Fanuc TP program (LS listing): JOB_VAR_SETUP.LS

/PROG  JOB_VAR_SETUP
/ATTR
OWNER		= MNEDITOR;
COMMENT		= "";
PROG_SIZE	= 12065;
CREATE		= DATE 19-06-21  TIME 11:36:36;
MODIFIED	= DATE 25-04-24  TIME 17:11:18;
FILE_NAME	= JOB_VAR_;
VERSION		= 0;
LINE_COUNT	= 453;
MEMORY_SIZE	= 12577;
PROTECT		= READ_WRITE;
TCD:  STACK_SIZE	= 0,
      TASK_PRIORITY	= 50,
      TIME_SLICE	= 0,
      BUSY_LAMP_OFF	= 0,
      ABORT_REQUEST	= 0,
      PAUSE_REQUEST	= 0;
DEFAULT_GROUP	= 1,*,*,*,*;
CONTROL_CODE	= 00000000 00000000;
/APPL

AUTO_SINGULARITY_HEADER;
  ENABLE_SINGULARITY_AVOIDANCE   : TRUE;
/MN
   1:  !--------------------------- ;
   2:  !Define the following run-time ;
   3:  !System variables, based on specs ;
   4:  !R[105]=AR[1]=100, 2By3 Sheet ;
   5:  !R[105]=AR[1]=200, 3By4 Sheet ;
   6:  !R[105]=AR[1]=300, 5By7 Sheet ;
   7:  !R[105]=AR[1]=400, 4By6 Sheet ;
   8:  !--------------------------- ;
   9:  !Input AR[1] Determines Setup ;
  10:  R[105]=AR[1]    ;
  11:  SELECT R[105]=100,JMP LBL[100] ;
  12:  !--------------------------- ;
  13:  !3By4 Sheet, 36 piece per Infeed ;
  14:  !Table Point, 36 Per level ;
  15:  !--------------------------- ;
  16:         =200,JMP LBL[200] ;
  17:  !--------------------------- ;
  18:  !3By4 Sheet Mandrel, 36 piece per ;
  19:  !Table Point, 36 Per level ;
  20:  !--------------------------- ;
  21:         =210,JMP LBL[210] ;
  22:  !--------------------------- ;
  23:  !3By4 , 36 piece per ;
  24:  !BOX, 36 Per level ;
  25:  !--------------------------- ;
  26:         =220,JMP LBL[220] ;
  27:  !--------------------------- ;
  28:  !5By7 Sheet, 35 piece per tray ;
  29:  !Table Point, 35 Per tray ;
  30:  !--------------------------- ;
  31:         =300,JMP LBL[300] ;
  32:  !--------------------------- ;
  33:  !4By6 INF, 144 piece per table ;
  34:  !4By9 OTF, 144 piece per table ;
  35:  !--------------------------- ;
  36:         =400,JMP LBL[400] ;
  37:  !--------------------------- ;
  38:  !Bar Feed, Outfeed Only ;
  39:  !4By9 OTF, 144 piece per table ;
  40:  !--------------------------- ;
  41:         =410,JMP LBL[410] ;
  42:  !--------------------------- ;
  43:  !4By6 INF, 144 piece per table ;
  44:  !6By8 OTF, 144 piece per table ;
  45:  !--------------------------- ;
  46:         =450,JMP LBL[450] ;
  47:  !--------------------------- ;
  48:  !6By8 OTF, 144 piece per table ;
  49:  !--------------------------- ;
  50:         =470,JMP LBL[470] ;
  51:  !--------------------------- ;
  52:  !3By4 Sheet, metal plate 12 piece ;
  53:  !Table Point, 36 Per tray ;
  54:  !--------------------------- ;
  55:         =500,JMP LBL[500] ;
  56:  !--------------------------- ;
  57:  !3By4 Sheet, 12 piece per tray ;
  58:  !Table Point, 72 Per level ;
  59:  !--------------------------- ;
  60:         =600,JMP LBL[600] ;
  61:  !--------------------------- ;
  62:  !Pallet data from Karel program ;
  63:  !--------------------------- ;
  64:         =900,JMP LBL[900] ;
  65:  !--------------------------- ;
  66:  !Beginning of Logic Program ;
  67:  !--------------------------- ;
  68:  LBL[100] ;
  69:  !--------------------------- ;
  70:  !2By3 Sheet, 6 piece per Infeed ;
  71:  !Table Point, 18 Per level ;
  72:  !--------------------------- ;
  73:  !1st: Infeed Row Offset ;
  74:  R[80]=191    ;
  75:  !2nd: Infeed Column Offset ;
  76:  R[81]=191    ;
  77:  !3rd: Infeed Division Offset ;
  78:  R[82]=2    ;
  79:  !4th: Infeed Modulus Offset ;
  80:  R[83]=2    ;
  81:  !5th: Infeed # of Pieces Per ;
  82:  !P[1], ie. One Level 3*(#) ;
  83:  !P[1] segnment of table, R[84] ;
  84:  R[84]=18    ;
  85:  !6th: Outfeed Row Offset ;
  86:  R[90]=191    ;
  87:  !7th: Outfeed Column Offset ;
  88:  R[91]=191    ;
  89:  !8th: Outfeed Division Offset ;
  90:  R[92]=2    ;
  91:  !9th: Outfeed Modulus Offset ;
  92:  R[93]=2    ;
  93:  !10th: Outfeed # of Pieces Per ;
  94:  !P[1], ie. One Level 3*(#) ;
  95:  !P[1] segnment of table, R[94] ;
  96:  R[94]=18    ;
  97:  JMP LBL[5000] ;
  98:   ;
  99:  LBL[200] ;
 100:  !--------------------------- ;
 101:  !3By4 Sheet, 12 piece per Infeed ;
 102:  !Table Point, 36 Per level ;
 103:  !--------------------------- ;
 104:  !1st: Infeed Row Offset ;
 105:  R[80]=140    ;
 106:  !2nd: Infeed Column Offset ;
 107:  R[81]=140    ;
 108:  !3rd: Infeed Division Offset ;
 109:  R[82]=3    ;
 110:  !4th: Infeed Modulus Offset ;
 111:  R[83]=3    ;
 112:  !5th: Infeed # of Pieces Per ;
 113:  !P[1], ie. One Level 3*(#) ;
 114:  !P[1] segnment of table, R[84] ;
 115:  R[84]=36    ;
 116:  !6th: Outfeed Row Offset ;
 117:  R[90]=130    ;
 118:  !7th: Outfeed Column Offset ;
 119:  R[91]=130    ;
 120:  !8th: Outfeed Division Offset ;
 121:  R[92]=3    ;
 122:  !9th: Outfeed Modulus Offset ;
 123:  R[93]=3    ;
 124:  !10th: Outfeed # of Pieces Per ;
 125:  !P[1], ie. One Level 3*(#) ;
 126:  !P[1] segnment of table, R[94] ;
 127:  R[94]=36    ;
 128:  JMP LBL[5000] ;
 129:   ;
 130:  LBL[210] ;
 131:  !--------------------------- ;
 132:  !3By4 Sheet, 12 piece per Infeed ;
 133:  !Table Point, 36 Per level ;
 134:  !metal plate, for mandrel ;
 135:  !--------------------------- ;
 136:  !1st: Infeed Row Offset ;
 137:  R[80]=126.9    ;
 138:  !2nd: Infeed Column Offset ;
 139:  R[81]=126.8    ;
 140:  !3rd: Infeed Division Offset ;
 141:  R[82]=3    ;
 142:  !4th: Infeed Modulus Offset ;
 143:  R[83]=3    ;
 144:  !5th: Infeed # of Pieces Per ;
 145:  !P[1], ie. One Level 3*(#) ;
 146:  !P[1] segnment of table, R[84] ;
 147:  R[84]=36    ;
 148:  !6th: Outfeed Row Offset ;
 149:  R[90]=130    ;
 150:  !7th: Outfeed Column Offset ;
 151:  R[91]=131    ;
 152:  !8th: Outfeed Division Offset ;
 153:  R[92]=3    ;
 154:  !9th: Outfeed Modulus Offset ;
 155:  R[93]=3    ;
 156:  !10th: Outfeed # of Pieces Per ;
 157:  !P[1], ie. One Level 3*(#) ;
 158:  !P[1] segnment of table, R[94] ;
 159:  R[94]=36    ;
 160:  JMP LBL[5000] ;
 161:  !--------------------------- ;
 162:  LBL[220] ;
 163:  !--------------------------- ;
 164:  !3By4 BOX, 12 piece per Infeed ;
 165:  !Table Point, 36 Per level ;
 166:  !--------------------------- ;
 167:  !1st: Infeed Row Offset ;
 168:  R[80]=127.2    ;
 169:  !2nd: Infeed Column Offset ;
 170:  R[81]=128.1    ;
 171:  !3rd: Infeed Division Offset ;
 172:  R[82]=3    ;
 173:  !4th: Infeed Modulus Offset ;
 174:  R[83]=3    ;
 175:  !5th: Infeed # of Pieces Per ;
 176:  !P[1], ie. One Level 3*(#) ;
 177:  !P[1] segnment of table, R[84] ;
 178:  R[84]=36    ;
 179:  !6th: Outfeed Row Offset ;
 180:  R[90]=127    ;
 181:  !7th: Outfeed Column Offset ;
 182:  R[91]=127    ;
 183:  !8th: Outfeed Division Offset ;
 184:  R[92]=3    ;
 185:  !9th: Outfeed Modulus Offset ;
 186:  R[93]=3    ;
 187:  !10th: Outfeed # of Pieces Per ;
 188:  !P[1], ie. One Level 3*(#) ;
 189:  !P[1] segnment of table, R[94] ;
 190:  R[94]=36    ;
 191:  JMP LBL[5000] ;
 192:   ;
 193:  LBL[300] ;
 194:  !--------------------------- ;
 195:  !5By7 Sheet, 35 piece per Infeed ;
 196:  !Table Point, 105 Per level ;
 197:  !--------------------------- ;
 198:  !1st: Infeed Row Offset ;
 199:  R[80]=76.2    ;
 200:  !2nd: Infeed Column Offset ;
 201:  R[81]=76.2    ;
 202:  !3rd: Infeed Division Offset ;
 203:  R[82]=5    ;
 204:  !4th: Infeed Modulus Offset ;
 205:  R[83]=5    ;
 206:  !5th: Infeed # of Pieces Per ;
 207:  !P[1], ie. One Level 3*(#) ;
 208:  !P[1] segnment of table, R[84] ;
 209:  R[84]=105    ;
 210:  !6th: Outfeed Row Offset ;
 211:  R[90]=130    ;
 212:  !7th: Outfeed Column Offset ;
 213:  R[91]=130    ;
 214:  !8th: Outfeed Division Offset ;
 215:  R[92]=3    ;
 216:  !9th: Outfeed Modulus Offset ;
 217:  R[93]=3    ;
 218:  !10th: Outfeed # of Pieces Per ;
 219:  !P[1], ie. One Level 3*(#) ;
 220:  !P[1] segnment of table, R[94] ;
 221:  R[94]=36    ;
 222:  JMP LBL[5000] ;
 223:   ;
 224:  LBL[400] ;
 225:  !--------------------------- ;
 226:  !4By6 INF, 24 piece per tray, 144 ;
 227:  !4By9 OTF, 36 piece per tray, 144 ;
 228:  !--------------------------- ;
 229:  !1st: Infeed Row Offset ;
 230:  R[80]=101.6    ;
 231:  !2nd: Infeed Column Offset ;
 232:  R[81]=101.8    ;
 233:  !3rd: Infeed Division Offset ;
 234:  R[82]=4    ;
 235:  !4th: Infeed Modulus Offset ;
 236:  R[83]=4    ;
 237:  !5th: Infeed # of Pieces Per ;
 238:  !P[1], ie. One Level 3*(#) ;
 239:  !P[1] segnment of table, R[84] ;
 240:  R[84]=144    ;
 241:  !6th: Outfeed Row Offset ;
 242:  R[90]=63.5    ;
 243:  !7th: Outfeed Column Offset ;
 244:  R[91]=63    ;
 245:  !8th: Outfeed Division Offset ;
 246:  R[92]=4    ;
 247:  !9th: Outfeed Modulus Offset ;
 248:  R[93]=4    ;
 249:  !10th: Outfeed # of Pieces Per ;
 250:  !P[1], ie. One Level 3*(#) ;
 251:  !P[1] segnment of table, R[94] ;
 252:  R[94]=144    ;
 253:  JMP LBL[5000] ;
 254:   ;
 255:  LBL[410] ;
 256:  !--------------------------- ;
 257:  !4By9 OTF, 36 piece per tray, 144 ;
 258:  !--------------------------- ;
 259:  !1st: Infeed Row Offset ;
 260:  R[80]=101.6    ;
 261:  !2nd: Infeed Column Offset ;
 262:  R[81]=101.8    ;
 263:  !3rd: Infeed Division Offset ;
 264:  R[82]=4    ;
 265:  !4th: Infeed Modulus Offset ;
 266:  R[83]=4    ;
 267:  !5th: Infeed # of Pieces Per ;
 268:  !P[1], ie. One Level 3*(#) ;
 269:  !P[1] segnment of table, R[84] ;
 270:  R[84]=144    ;
 271:  !6th: Outfeed Row Offset ;
 272:  R[90]=63.5    ;
 273:  !7th: Outfeed Column Offset ;
 274:  R[91]=63.5    ;
 275:  !8th: Outfeed Division Offset ;
 276:  R[92]=4    ;
 277:  !9th: Outfeed Modulus Offset ;
 278:  R[93]=4    ;
 279:  !10th: Outfeed # of Pieces Per ;
 280:  !P[1], ie. One Level 3*(#) ;
 281:  !P[1] segnment of table, R[94] ;
 282:  R[94]=144    ;
 283:  JMP LBL[5000] ;
 284:   ;
 285:  LBL[450] ;
 286:  !--------------------------- ;
 287:  !4By6 INF, 24 piece per tray, 144 ;
 288:  !6By8 OTF, 48 piece per tray, 144 ;
 289:  !--------------------------- ;
 290:  !1st: Infeed Row Offset ;
 291:  R[80]=101.6    ;
 292:  !2nd: Infeed Column Offset ;
 293:  R[81]=101.8    ;
 294:  !3rd: Infeed Division Offset ;
 295:  R[82]=4    ;
 296:  !4th: Infeed Modulus Offset ;
 297:  R[83]=4    ;
 298:  !5th: Infeed # of Pieces Per ;
 299:  !P[1], ie. One Level 3*(#) ;
 300:  !P[1] segnment of table, R[84] ;
 301:  R[84]=144    ;
 302:  !6th: Outfeed Row Offset ;
 303:  R[90]=65    ;
 304:  !7th: Outfeed Column Offset ;
 305:  R[91]=65    ;
 306:  !8th: Outfeed Division Offset ;
 307:  R[92]=8    ;
 308:  !9th: Outfeed Modulus Offset ;
 309:  R[93]=8    ;
 310:  !10th: Outfeed # of Pieces Per ;
 311:  !P[1], ie. One Level 3*(#) ;
 312:  !P[1] segnment of table, R[94] ;
 313:  R[94]=144    ;
 314:  JMP LBL[5000] ;
 315:   ;
 316:  LBL[470] ;
 317:  !--------------------------- ;
 318:  !4By6 INF, 24 piece per tray, 144 ;
 319:  !6By8 OTF, 48 piece per tray, 144 ;
 320:  !--------------------------- ;
 321:  !1st: Infeed Row Offset ;
 322:  R[80]=101.6    ;
 323:  !2nd: Infeed Column Offset ;
 324:  R[81]=101.8    ;
 325:  !3rd: Infeed Division Offset ;
 326:  R[82]=4    ;
 327:  !4th: Infeed Modulus Offset ;
 328:  R[83]=4    ;
 329:  !5th: Infeed # of Pieces Per ;
 330:  !P[1], ie. One Level 3*(#) ;
 331:  !P[1] segnment of table, R[84] ;
 332:  R[84]=144    ;
 333:  !6th: Outfeed Row Offset ;
 334:  R[90]=60    ;
 335:  !7th: Outfeed Column Offset ;
 336:  R[91]=60    ;
 337:  !8th: Outfeed Division Offset ;
 338:  R[92]=6    ;
 339:  !9th: Outfeed Modulus Offset ;
 340:  R[93]=6    ;
 341:  !10th: Outfeed # of Pieces Per ;
 342:  !P[1], ie. One Level 3*(#) ;
 343:  !P[1] segnment of table, R[94] ;
 344:  R[94]=144    ;
 345:  JMP LBL[5000] ;
 346:   ;
 347:  LBL[500] ;
 348:  !--------------------------- ;
 349:  !3By4 Sheet, metal plate 12 piece ;
 350:  !Table Point, 36 Per level ;
 351:  !--------------------------- ;
 352:  !1st: Infeed Row Offset ;
 353:  R[80]=126.3    ;
 354:  !2nd: Infeed Column Offset ;
 355:  R[81]=126.8    ;
 356:  !3rd: Infeed Division Offset ;
 357:  R[82]=3    ;
 358:  !4th: Infeed Modulus Offset ;
 359:  R[83]=3    ;
 360:  !5th: Infeed # of Pieces Per ;
 361:  !P[1], ie. One Level 3*(#) ;
 362:  !P[1] segnment of table, R[84] ;
 363:  R[84]=36    ;
 364:  !6th: Outfeed Row Offset ;
 365:  R[90]=130    ;
 366:  !7th: Outfeed Column Offset ;
 367:  R[91]=132    ;
 368:  !8th: Outfeed Division Offset ;
 369:  R[92]=3    ;
 370:  !9th: Outfeed Modulus Offset ;
 371:  R[93]=3    ;
 372:  !10th: Outfeed # of Pieces Per ;
 373:  !P[1], ie. One Level 3*(#) ;
 374:  !P[1] segnment of table, R[94] ;
 375:  R[94]=36    ;
 376:  JMP LBL[5000] ;
 377:   ;
 378:  LBL[600] ;
 379:  !--------------------------- ;
 380:  !3By4 Sheet, 12 piece per tray ;
 381:  !Table Point, 72 Per level ;
 382:  !--------------------------- ;
 383:  !1st: Infeed Row Offset ;
 384:  R[80]=140    ;
 385:  !2nd: Infeed Column Offset ;
 386:  R[81]=140    ;
 387:  !3rd: Infeed Division Offset ;
 388:  R[82]=3    ;
 389:  !4th: Infeed Modulus Offset ;
 390:  R[83]=3    ;
 391:  !5th: Infeed # of Pieces Per ;
 392:  !P[1], ie. One Level 3*(#) ;
 393:  !P[1] segnment of table, R[84] ;
 394:  R[84]=72    ;
 395:  !6th: Outfeed Row Offset ;
 396:  R[90]=140    ;
 397:  !7th: Outfeed Column Offset ;
 398:  R[91]=140    ;
 399:  !8th: Outfeed Division Offset ;
 400:  R[92]=2    ;
 401:  !9th: Outfeed Modulus Offset ;
 402:  R[93]=2    ;
 403:  !10th: Outfeed # of Pieces Per ;
 404:  !P[1], ie. One Level 3*(#) ;
 405:  !P[1] segnment of table, R[94] ;
 406:  R[94]=32    ;
 407:  JMP LBL[5000] ;
 408:   ;
 409:  LBL[900] ;
  410:  !--------------------------- ;
 411:  !Pallet data from Karel program ;
 412:  !--------------------------- ;
 413:  CALL GN_CLS_SC_F9 ;
 414:  MESSAGE[PALLET data is loading.] ;
 415:  WAIT 1.00(sec) ;
 416:  !1st: Infeed Row Spacing ;
 417:  R[80]=R[424] ;
 418:  !2nd: Infeed Column Spacing ;
 419:  R[81]=R[425] ;
 420:  !3rd: Division - column count ;
 421:  R[82]=R[423] ;
 422:  !4th: Modulus - column count ;
 423:  R[83]=R[423] ;
 424:  !5th: Infeed whole-table slots ;
 425:  !PALLET_SLOTS is total on table ;
 426:  !Use loaded pallet slot count ;
 427:  R[84]=R[427] ;
 428:  !6th: Outfeed Row Spacing ;
 429:  R[90]=R[424] ;
 430:  !7th: Outfeed Column Spacing ;
 431:  R[91]=R[425] ;
 432:  !8th: Division - column count ;
 433:  R[92]=R[423] ;
 434:  !9th: Modulus - column count ;
 435:  R[93]=R[423] ;
 436:  !10th: Outfeed whole-table slots ;
 437:  !Same capacity as infeed ;
 438:  !Use loaded pallet slot count ;
 439:  R[94]=R[427] ;
 440:  JMP LBL[5000] ;
 441:   ;
 442:  !--------------------------- ;
 443:  LBL[5000] ;
 444:  !--------------------------- ;
 445:  !This program assigns the values ;
 446:  !Into correct register for usuage ;
 447:  !--------------------------- ;
 448:  CALL CREATE_OFFSETS(R[80],R[81],R[82],R[83],R[84],R[90],R[91],R[92],R[93],R[94]) ;
 449:  !--------------------------- ;
 450:  JMP LBL[9999] ;
 451:  !--------------------------- ;
 452:  LBL[9999:END] ;
 453:  END ;
/POS
/END
